// TwinCAT 3 PLC project PLC1
// ProgramVersion: 3.1.4024.0
// libraries:
//   SPT Base Types, * (Beckhoff Automation LLC)
//   SPT Event Logger, * (Beckhoff Automation LLC)
//   Tc2_Standard, * (Beckhoff Automation GmbH)
//   Tc2_System, * (Beckhoff Automation GmbH)
//   Tc3_Module, * (Beckhoff Automation GmbH)
//   XPlanarApplication, * (Beckhoff Automation LLC)
// project tree:
//   / GlobalTextList.TcGTLO, PlcTask.TcTTO, Visualization Manager.TcVMO (not stored)
//   POUs/CustomStations/ FB_RoutingStation.TcPOU, FB_RotateStation.TcPOU
//   POUs/ FB_XPlanarModule.TcPOU, MAIN.TcPOU
//   POUs/Utilities/ ErrorStep.TcPOU (not stored), NextMinorStep.TcPOU (not stored), NextStep.TcPOU
//   VISUs/ V_Main.TcVIS
// real-time tasks:
//   TASK XPlanar Task3: cycle T#250us, priority 1, ADS port 350
//   TASK XPlanar Task4: cycle T#250us, priority 2, ADS port 351
//   TASK XPlanar Task5: cycle T#250us, priority 3, ADS port 352
//   TASK MC-Task (MET): cycle T#2ms, priority 4, ADS port 353
//   TASK MC-Task (MPT): cycle T#10ms, priority 5, ADS port 354
//   TASK Job Task: cycle default, priority 6
//   TASK PlcTask: cycle T#10ms, priority 20, ADS port 355
// variable links:
//   XPlanar MC Project/Axes/Mover4330_1 <-> TcCOM Objects/XPlanar/Mover4330_1
//     McToIo/STD <-> InputsFromNC3/NC3ToHW
//   XPlanar MC Project/Axes/Mover4330_2 <-> TcCOM Objects/XPlanar/Mover4330_2
//     IoToMc/STD <-> OutputsToNC3/HWToNC3
//   XPlanar MC Project/Axes/Mover4330_3 <-> TcCOM Objects/XPlanar/Mover4330_3
//     IoToMc/STD <-> OutputsToNC3/HWToNC3
//   XPlanar MC Project/Axes/Mover4330_4 <-> TcCOM Objects/XPlanar/Mover4330_4
//     IoToMc/STD <-> OutputsToNC3/HWToNC3
//   PLC1/PLC1 Instance <-> XPlanar MC Project/Axes/Mover4330_1
//     PlcTask Inputs/MAIN.XPlanarModule.Mover[1]._Mover.MCTOPLC/ACT <-> McToPlc/ACT
//     PlcTask Inputs/MAIN.XPlanarModule.Mover[1]._Mover.MCTOPLC/COORDMODE <-> McToPlc/COORDMODE
//     PlcTask Inputs/MAIN.XPlanarModule.Mover[1]._Mover.MCTOPLC/SET <-> McToPlc/SET
//     PlcTask Inputs/MAIN.XPlanarModule.Mover[1]._Mover.MCTOPLC/SETONTRACK <-> McToPlc/SETONTRACK
//     PlcTask Inputs/MAIN.XPlanarModule.Mover[1]._Mover.MCTOPLC/STD <-> McToPlc/STD
//     PlcTask Outputs/MAIN.XPlanarModule.Mover[1]._Mover.PLCTOMC/STD <-> PlcToMc/STD
//   PLC1/PLC1 Instance <-> XPlanar MC Project/Axes/Mover4330_2
//     PlcTask Inputs/MAIN.XPlanarModule.Mover[2]._Mover.MCTOPLC/ACT <-> McToPlc/ACT
//     PlcTask Inputs/MAIN.XPlanarModule.Mover[2]._Mover.MCTOPLC/COORDMODE <-> McToPlc/COORDMODE
//     PlcTask Inputs/MAIN.XPlanarModule.Mover[2]._Mover.MCTOPLC/SET <-> McToPlc/SET
//     PlcTask Inputs/MAIN.XPlanarModule.Mover[2]._Mover.MCTOPLC/SETONTRACK <-> McToPlc/SETONTRACK
//     PlcTask Inputs/MAIN.XPlanarModule.Mover[2]._Mover.MCTOPLC/STD <-> McToPlc/STD
//     PlcTask Outputs/MAIN.XPlanarModule.Mover[2]._Mover.PLCTOMC/STD <-> PlcToMc/STD
//   PLC1/PLC1 Instance <-> XPlanar MC Project/Axes/Mover4330_3
//     PlcTask Inputs/MAIN.XPlanarModule.Mover[3]._Mover.MCTOPLC/ACT <-> McToPlc/ACT
//     PlcTask Inputs/MAIN.XPlanarModule.Mover[3]._Mover.MCTOPLC/COORDMODE <-> McToPlc/COORDMODE
//     PlcTask Inputs/MAIN.XPlanarModule.Mover[3]._Mover.MCTOPLC/SET <-> McToPlc/SET
//     PlcTask Inputs/MAIN.XPlanarModule.Mover[3]._Mover.MCTOPLC/SETONTRACK <-> McToPlc/SETONTRACK
//     PlcTask Inputs/MAIN.XPlanarModule.Mover[3]._Mover.MCTOPLC/STD <-> McToPlc/STD
//     PlcTask Outputs/MAIN.XPlanarModule.Mover[3]._Mover.PLCTOMC/STD <-> PlcToMc/STD
//   PLC1/PLC1 Instance <-> XPlanar MC Project/Axes/Mover4330_4
//     PlcTask Inputs/MAIN.XPlanarModule.Mover[4]._Mover.MCTOPLC/ACT <-> McToPlc/ACT
//     PlcTask Inputs/MAIN.XPlanarModule.Mover[4]._Mover.MCTOPLC/COORDMODE <-> McToPlc/COORDMODE
//     PlcTask Inputs/MAIN.XPlanarModule.Mover[4]._Mover.MCTOPLC/SET <-> McToPlc/SET
//     PlcTask Inputs/MAIN.XPlanarModule.Mover[4]._Mover.MCTOPLC/SETONTRACK <-> McToPlc/SETONTRACK
//     PlcTask Inputs/MAIN.XPlanarModule.Mover[4]._Mover.MCTOPLC/STD <-> McToPlc/STD
//     PlcTask Outputs/MAIN.XPlanarModule.Mover[4]._Mover.PLCTOMC/STD <-> PlcToMc/STD
//   PLC1/PLC1 Instance <-> XPlanar MC Project/Groups/Environment
//     PlcTask Inputs/XPlanarApplication.XPlanar.Environment.MCTOPLC_STD <-> McToPlc/STD
//   PLC1/PLC1 Instance <-> XPlanar MC Project/Groups/Track1
//     PlcTask Inputs/MAIN.XPlanarModule.Track[1]._Track.MCTOPLC_STD <-> McToPlc/STD
//   PLC1/PLC1 Instance <-> XPlanar MC Project/Groups/Track2
//     PlcTask Inputs/MAIN.XPlanarModule.Track[2]._Track.MCTOPLC_STD <-> McToPlc/STD
//   PLC1/PLC1 Instance <-> XPlanar MC Project/Groups/Track3
//     PlcTask Inputs/MAIN.XPlanarModule.Track[3]._Track.MCTOPLC_STD <-> McToPlc/STD
//   PLC1/PLC1 Instance <-> XPlanar MC Project/Groups/XPlanar
//     PlcTask Inputs/XPlanarApplication.XPlanar.Group.MCTOPLC_STD <-> McToPlc/STD
//   TcCOM Objects/XPlanar/Mover4330_1 <-> XPlanar MC Project/Axes/Mover4330_1
//     OutputsToNC3/HWToNC3 <-> IoToMc/STD
//   TcCOM Objects/XPlanar/Mover4330_2 <-> XPlanar MC Project/Axes/Mover4330_2
//     InputsFromNC3/NC3ToHW <-> McToIo/STD
//   TcCOM Objects/XPlanar/Mover4330_3 <-> XPlanar MC Project/Axes/Mover4330_3
//     InputsFromNC3/NC3ToHW <-> McToIo/STD
//   TcCOM Objects/XPlanar/Mover4330_4 <-> XPlanar MC Project/Axes/Mover4330_4
//     InputsFromNC3/NC3ToHW <-> McToIo/STD

CONFIGURATION PLC1
    RESOURCE PLC ON TwinCAT3
        TASK PlcTask(INTERVAL := T#10ms, PRIORITY := 20);
        PROGRAM MAIN WITH PlcTask : MAIN;
    END_RESOURCE
END_CONFIGURATION

// ---- POUs/MAIN.TcPOU
PROGRAM MAIN
VAR
	//Main machine module declaration
	XPlanarModule : FB_XPlanarModule;

	//Control Source for running machine
	ControlSourceHMI : FB_ControlSource;
	ControlSourcePB	 : FB_ControlSource;

	//Local Vars
	InitComplete : BOOL;
END_VAR

CyclicLogic();

METHOD CyclicLogic
VAR_INPUT
END_VAR
IF NOT InitComplete THEN
	InitComplete := Initialize();
	RETURN;
END_IF

//Machine support HMI & Production Monitor
ControlSourcePB.CyclicLogic();
ControlSourceHMI.CyclicLogic();

//Machine Cyclic Logic
XPlanarModule.CyclicLogic();
END_METHOD

METHOD Initialize : BOOL
//Top level machine initialization should happen here, in the main initialization METHOD. Each subsequent "layer" OF modules will be named within their respective "parent" intialize METHOD
IF NOT ControlSourceHMI.Registered THEN
	XPlanarModule.RegisterExternalController(ControlSourceHMI);
END_IF

IF NOT ControlSourcePB.Registered THEN
	XPlanarModule.RegisterExternalController(ControlSourcePB);
END_IF

ControlSourceHMI.CyclicLogic();
ControlSourcePB.CyclicLogic();

//ADSLOGSTR(ADSLOG_MSGTYPE_WARN, 'Lag Monitoring disabled', 'For simulation demo only',);
Initialize := TRUE;
END_METHOD

END_PROGRAM

// ---- POUs/FB_XPlanarModule.TcPOU
FUNCTION_BLOCK FB_XPlanarModule EXTENDS FB_PackML_BaseModule
VAR
	// Component definitions here
	XPlanarTable : FB_Component_Xplanar := (Name := 'XPlanarTable');

	//Station Components
	Station1 : FB_RotateStation	 := (Name := 'Station1'); //Declaration of a custom station
	Station2 : FB_RoutingStation := (Name := 'Station2');
	Station3 : FB_RotateStation	 := (Name := 'Station3');
	Station4 : FB_RotateStation	 := (Name := 'Station4');

	//Helper Vars
	Mover			  : ARRAY[1..SystemParameters.MOVER_COUNT] OF FB_XPlanarMover;
	Track			  : ARRAY[1..SystemParameters.TRACK_COUNT] OF FB_XPlanarTrackSegment;
	TracksInitialized : BOOL;
END_VAR

//! @summary This method contains code which will execute when this PackML module is in the <b>Aborting</b> state
METHOD PROTECTED Aborting
VAR
	i				: UDINT;
	SubModulesReady : BOOL := TRUE;
END_VAR
CASE DescendantSequenceState OF
	0:
		NoStateTasksToComplete := FALSE;
		NextStep(DescendantSequenceState);

	10:
		IF XPlanarTable.Abort() THEN
			StateTasksComplete := TRUE;
			NextStep(DescendantSequenceState);
		END_IF

	20:
		StateTasksComplete := TRUE;
END_CASE

SUPER^.Aborting();
END_METHOD

//! @summary This method contains code which will execute when this PackML module is in the <b>Clearing</b> state
METHOD PROTECTED Clearing
VAR
	i				: UDINT;
	SubModulesReady : BOOL := TRUE;
END_VAR

VAR_INST
	ipResult : I_PlanarTaskResult;
END_VAR

(*! <description> <b>Note:</b> The <i>Clear</i> command can also be thought of as a <i>fault reset</i> depite the ambiguity in the naming of the <i>Reset</i> state. 
<table> 
	<tr>
		<th> Previous State </th>
		<th> Transition In </th>
		<th> Transition Out </th>
		<th> Next State  </th> 
	</tr>
	<tr>
		<td> Aborted </td>
		<td> Clear Command </td> 
		<td> State Complete </td>
		<td> Stopped </td> 
	</tr>
</table>
This method is called as required by <c>StateControl()</c>
</description> 

*)
CASE _CurrentMode OF
	E_PMLUnitMode.ePMLUnitMode_Production:
		CASE DescendantSequenceState OF
			0: //Init
				NoStateTasksToComplete := FALSE;

				//Reset Stations
				Station1.Reset();
				Station2.Reset();
				Station3.Reset();
				NextStep(DescendantSequenceState);

			10: //Reset XPlanar System
				IF XPlanarTable.Reset() THEN
					NextStep(DescendantSequenceState);
				END_IF

			20: //Enable Group
				ipResult := XPlanarTable.EnableGroup();
				IF ipResult.Done THEN
					NextStep(DescendantSequenceState);
				ELSIF ipResult.Error THEN
					ErrorStep(DescendantSequenceState);
				END_IF

			30: //Clearing complete			
				StateTasksComplete := TRUE;
		END_CASE

	E_PMLUnitMode.ePMLUnitMode_Manual:
		;
END_CASE

SUPER^.Clearing();
END_METHOD

METHOD CyclicLogic
VAR
	i : INT;
END_VAR
IF NOT _InitComplete THEN
	_InitComplete := Initialize();
END_IF

//Add any required cyclic logic here

//Call the base logic
SUPER^.CyclicLogic();
END_METHOD

//! @summary This method contains code which will execute when this PackML module is in the <b>Execute</b> state
METHOD PROTECTED Execute
VAR
	i : UDINT;
END_VAR
CASE _CurrentMode OF
	E_PMLUnitMode.ePMLUnitMode_Production:
		FOR i := 1 TO SystemParameters.STATION_COUNT DO
			ip.Stations[i].Execute();
		END_FOR

	E_PMLUnitMode.ePMLUnitMode_Manual:
		; //Insert logic for Manual Mode here
END_CASE
END_METHOD

//! @summary Automatically enables and disables HMI control based on the PackML mode
METHOD PROTECTED HMIPermissions

//! @description This method is called cyclically by <c>CyclicLogic()</c>
//General Mode Based Monitoring and handling of HMI control
CASE _CurrentMode OF
	E_PMLUnitMode.ePMLUnitMode_Production:
		AllowHMIControl(ThisModuleOnly := FALSE);

	E_PMLUnitMode.ePMLUnitMode_Manual:
		AllowHMIControl(ThisModuleOnly := FALSE);

	E_PMLUnitMode.ePMLUnitMode_Maintenance:
		AllowHMIControl(ThisModuleOnly := FALSE);
END_CASE
END_METHOD

//! @summary Basic module initialization logic
METHOD PROTECTED Initialize : BOOL;
VAR
	i						 : UDINT;
	varInfo					 : __SYSTEM.VAR_INFO;
	AllSubUnitsInitialized	 : BOOL := TRUE;
	AllComponentsInitialized : BOOL := TRUE;
END_VAR

//! @description This method is called by <c>CyclicLogic()</c> as required
Initialize := FALSE;
CASE DescendantSequenceState OF
	0: //Register Submodules and Components
		RegisterComponent(XPlanarTable);
		RegisterComponent(Station1);
		RegisterComponent(Station2);
		RegisterComponent(Station3);
		RegisterComponent(Station4);
		_LogModeChanges			:= FALSE;
		_LogStateChanges		:= FALSE;
		DescendantSequenceState := DescendantSequenceState + 10;

	10: //Set interfaces *This must be done before initializing the base class!

		//Set mover interfaces
		FOR i := 1 TO SystemParameters.MOVER_COUNT DO
			Mover[i].MoverIndex := i;
			ip.Movers[i]		:= Mover[i];
		END_FOR

		//Set Track Interfaces
		FOR i := 1 TO SystemParameters.TRACK_COUNT DO
			ip.Tracks[i] := Track[i];
		END_FOR

		//Set Station interfaces
		ip.Stations[1]			:= Station1;
		ip.Stations[2]			:= Station2;
		ip.Stations[3]			:= Station3;
		ip.Stations[4]			:= Station4;
		DescendantSequenceState := DescendantSequenceState + 10;

	20: //Call Initialize of the base class
		IF SUPER^.Initialize() THEN
			DescendantSequenceState := DescendantSequenceState + 10;
		END_IF

	30:
		Initialize := TRUE;
END_CASE
END_METHOD

METHOD PROTECTED Resetting
VAR_INST
	i			 : UDINT;
	ipTaskResult : I_PlanarTaskResult;
END_VAR
CASE _CurrentMode OF
	E_PMLUnitMode.ePMLUnitMode_Production:
		CASE DescendantSequenceState OF
			0: //Init
				i					   := 1;
				NoStateTasksToComplete := FALSE;
				NextStep(DescendantSequenceState);

			10: //Enable Tracks
				ipTaskResult := XplanarTable.EnableTracks();
				IF ipTaskResult.Done THEN
					NextStep(DescendantSequenceState);
				ELSIF ipTaskResult.Error THEN //An error occured, jump to 'error step'
					ErrorStep(DescendantSequenceState);
				END_IF

			20: //Enable Movers
				ipTaskResult := XPlanarTable.EnableMovers();
				IF ipTaskResult.Done THEN
					NextStep(DescendantSequenceState);
				ELSIF ipTaskResult.Error THEN //An error occured, jump to 'error step'
					ErrorStep(DescendantSequenceState);
				END_IF

			30: //Add Tracks to Group
				ipTaskResult := XPlanarTable.AddTracksToGroup();
				IF ipTaskResult.Done THEN
					NextStep(DescendantSequenceState);
				ELSIF ipTaskResult.Error THEN //An error occured, jump to 'error step'
					ErrorStep(DescendantSequenceState);
				END_IF

			40: //Add Movers to Group			
				ipTaskResult := XPlanarTable.AddMoversToGroup();
				IF ipTaskResult.Done THEN
					NextStep(DescendantSequenceState);
				ELSIF ipTaskResult.Error THEN //An error occured, jump to 'error step'
					ErrorStep(DescendantSequenceState);
				END_IF

			50: //Clearing complete
				StateTasksComplete := TRUE;
		END_CASE
END_CASE

SUPER^.Resetting();
END_METHOD

METHOD PRIVATE SetupStations : BOOL
VAR_INPUT
END_VAR
//Set Required Process Station Initialization Parameters
Station1.Position.SetValuesXYC(120, 360, 0);
Station1.Size.x		   := 120;		//Changes the station size in the X plane (optional - Default is 120mm)
Station1.Size.y		   := 120;		//Changes the station size in the Y plane (optionsl- Default is 120mm)
Station1.TrackID	   := 1;		//Set Index of the track segment the station resides on if applicable	
Station1.NextStation   := Station2; //Set the interface for the next station of the mover
Station1.StationAngle  := 90;
Station1.NumberOfTurns := 0;

Station2.Position.SetValuesXYC(360, 600, 0);
Station2.StationType := E_StationType.DecisionPoint; //Set type to DecisionPoint for 'on the fly' processing
Station2.OutputA := Station3;
Station2.OutputB := Station4;
Station2.TrackID	   := 1;

Station3.Position.SetValuesXYC(600, 360, 0);
Station3.TrackID	   := 2;
Station3.NextStation   := Station1;
Station3.StationAngle  := 360;
Station3.NumberOfTurns := 1;

Station4.Position.SetValuesXYC(840, 360, 0);
Station4.TrackID	   := 3;
Station4.NextStation   := Station1;
Station4.StationAngle  := -90;
Station4.NumberOfTurns := 0;

//Return TRUE when all necessary station parameters are set
SetupStations := TRUE;
END_METHOD

METHOD PROTECTED Starting
VAR_INST
	i		 : UDINT;
	ipResult : I_PlanarTaskResult;
END_VAR
CASE _CurrentMode OF
	E_PMLUnitMode.ePMLUnitMode_Production:
		CASE DescendantSequenceState OF
			0:
				NoStateTasksToComplete	:= FALSE;
				DescendantSequenceState := 10;
				i						:= 1;

			10: //Set Station Parameters
				SetupStations();
				NextStep(DescendantSequenceState);

			20: //Cleanup mover queues
				FOR i := 1 TO SystemParameters.STATION_COUNT DO
					ip.Stations[i].MoverQueue.Dequeue();
				END_FOR

				NextStep(DescendantSequenceState);

			30: //Set some initial application move dynamics
				FOR i := 1 TO SystemParameters.MOVER_COUNT DO
					ip.Movers[i].Dynamics.Movement.Accel	:= 2000;
					ip.Movers[i].Dynamics.Movement.Decel	:= 2000;
					ip.Movers[i].Dynamics.Movement.Velocity := 300;
					ip.Movers[i].Dynamics.Movement.Jerk		:= 50000;
					ip.Movers[i].Dynamics.Rotation.Accel	:= 5000;
					ip.Movers[i].Dynamics.Rotation.Decel	:= 5000;
					ip.Movers[i].Dynamics.Rotation.Velocity := 300;
					ip.Movers[i].Dynamics.Rotation.Jerk		:= 100000;
					ip.Movers[i].Dynamics.Tilt.Accel		:= 5000;
					ip.Movers[i].Dynamics.Tilt.Decel		:= 5000;
					ip.Movers[i].Dynamics.Tilt.Velocity		:= 300;
					ip.Movers[i].Dynamics.Tilt.Jerk			:= 100000;
					ip.Movers[i].Gap						:= 250;
					ip.Movers[i].Destination				:= 0;
				END_FOR

				i := 1;
				NextStep(DescendantSequenceState);

			40: //Join Movers to nearest track
				IF i <= SystemParameters.MOVER_COUNT THEN
					ipResult := ip.Movers[i].MoveCommand.JoinClosestTrack(FALSE);
					IF ipResult.Done THEN
						NextMinorStep(DescendantSequenceState);
					ELSIF ipResult.Error THEN
						ErrorStep(DescendantSequenceState);
					END_IF
				ELSE
					i := 1;
					NextStep(DescendantSequenceState);
				END_IF

			41: //Check Mover Count
				IF i <= SystemParameters.MOVER_COUNT THEN
					i						:= i + 1;
					DescendantSequenceState := 40;
				ELSE
					i := 1;
					NextStep(DescendantSequenceState);
				END_IF

			50: //Send Movers around to station 1
				IF i <= SystemParameters.MOVER_COUNT THEN
					ipResult := ip.Movers[i].MoveCommand.SendToStation(ip.Stations[1]);
					IF ipResult.Busy THEN
						NextMinorStep(DescendantSequenceState);
					ELSIF ipResult.Error THEN
						ErrorStep(DescendantSequenceState);
					END_IF
				ELSE
					i := 1;
					NextStep(DescendantSequenceState);
				END_IF

			51: //Check Mover Count
				IF i <= SystemParameters.MOVER_COUNT THEN
					i						:= i + 1;
					DescendantSequenceState := 50;
				ELSE
					i := 1;
					NextStep(DescendantSequenceState);
				END_IF

			60:
				StateTasksComplete := TRUE;
		END_CASE

	E_PMLUnitMode.ePMLUnitMode_Manual:
		;
END_CASE

SUPER^.Starting();
END_METHOD

END_FUNCTION_BLOCK

// ---- POUs/CustomStations/FB_RotateStation.TcPOU
FUNCTION_BLOCK FB_RotateStation EXTENDS FB_XPlanarStationBase
VAR
	_StationAngle  : LREAL;
	_NumberOfTurns : DINT;
END_VAR

METHOD Execute
VAR_INST
	i			  : UDINT := 1;
	CommandResult : I_PlanarTaskResult;
END_VAR
SUPER^.Execute();
IF StationState = E_XPlanarStationState.ProcessMover THEN
	CommandResult := ipCurrentMover.MoveCommand.Rotate(_StationAngle, _NumberOfTurns);
	IF CommandResult.Done THEN
		_StationComplete := TRUE;
	ELSIF CommandResult.Error THEN
		; //Command returned an error!
	END_IF
END_IF
END_METHOD

PROPERTY NumberOfTurns : DINT
SET
_NumberOfTurns := NumberOfTurns;
END_SET
END_PROPERTY

PROPERTY StationAngle : LREAL
SET
_StationAngle := StationAngle;
END_SET
END_PROPERTY

END_FUNCTION_BLOCK

// ---- POUs/CustomStations/FB_RoutingStation.TcPOU
FUNCTION_BLOCK FB_RoutingStation EXTENDS FB_XPlanarStationBase
VAR_INPUT
END_VAR
VAR_OUTPUT
END_VAR
VAR
	_OutputA	: I_XplanarStation;
	_OutputB	: I_XPlanarStation;
END_VAR

METHOD Execute
SUPER^.Execute(); //Call the base station logic to handle sending and receiving of movers

//When the station is in the Process mover state you can perform any application specific station logic
IF StationState = E_XPlanarStationState.ProcessMover THEN
	IF _OutputA <> 0 AND _OutputB <> 0 THEN	
		CASE ipCurrentMover.MoverIndex OF
			1, 3:
				ipNextStation := _OutputA;
			2, 4:
				ipNextStation := _OutputB;
		END_CASE
		
		_StationComplete := TRUE;	//Set _StationComplete TRUE when done.  This will be automatically reset when the mover exits
	END_IF
END_IF
END_METHOD

PROPERTY OutputA : I_XPlanarStation
SET
_OutputA := OutputA;
END_SET
END_PROPERTY

PROPERTY OutputB : I_XPlanarStation
SET
_OutputB := OutputB;
END_SET
END_PROPERTY

END_FUNCTION_BLOCK

// ---- POUs/Utilities/NextStep.TcPOU
FUNCTION NextStep : UDINT
VAR_IN_OUT
	StateVar : UDINT;
END_VAR

NextStep := StateVar := ((StateVar / 10) * 10) + 10;

END_FUNCTION

// ---- GlobalTextList.TcGTLO
TEXTLIST GlobalTextList
  944 = 'HMI PB Station'
  924 = 'Pushbutton Station'
  181 = 'Reset'
  77 = 'Start'
  828 = 'Stop'
END_TEXTLIST

// ---- VISUs/V_Main.TcVIS
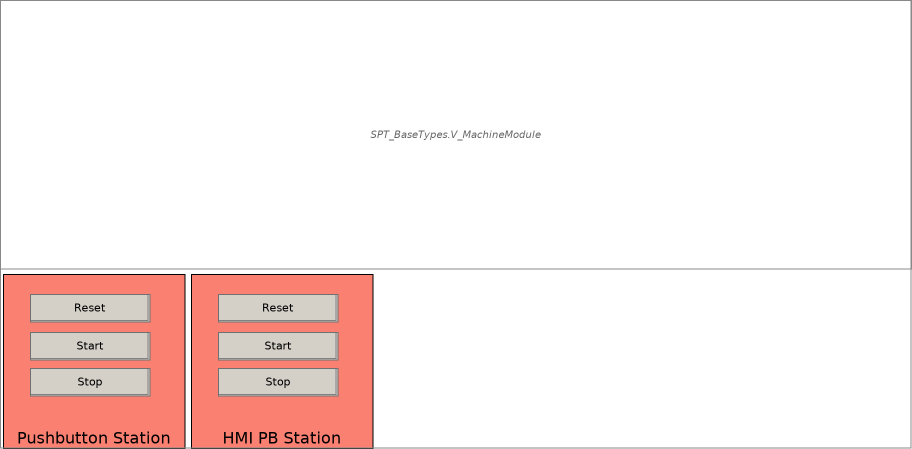
VISUALIZATION V_Main  // 912x449
    Frame (0,0 912x269)
        shows SPT_BaseTypes.V_MachineModule(HMI := MAIN.XPlanarModule.PackMLBaseModule_HMI)
    Group (3,274 182x175)
        RoundedRectangle (0,0 182x175), "Pushbutton Station"
        Button (27,94 120x28), "Stop", input disabled if: not MAIN.ControlSourcePB.MainPMLControl_Simplified.StopPermissive
            tap MAIN.ControlSourcePB.MainPMLControl_Simplified.StopPressed
        Button (27,20 120x28), "Reset", input disabled if: not MAIN.ControlSourcePB.MainPMLControl_Simplified.ResetPermissive
            tap MAIN.ControlSourcePB.MainPMLControl_Simplified.ResetPressed
        Button (27,58 120x28), "Start", input disabled if: not MAIN.ControlSourcePB.MainPMLControl_Simplified.StartPermissive
            tap MAIN.ControlSourcePB.MainPMLControl_Simplified.StartPressed
    Group (191,274 182x175)
        RoundedRectangle (0,0 182x175), "HMI PB Station"
        Button (27,94 120x28), "Stop", input disabled if: not MAIN.ControlSourceHMI.MainPMLControl_Simplified.StopPermissive
            tap MAIN.ControlSourceHMI.MainPMLControl_Simplified.StopPressed
        Button (27,20 120x28), "Reset", input disabled if: not MAIN.ControlSourceHMI.MainPMLControl_Simplified.ResetPermissive
            tap MAIN.ControlSourceHMI.MainPMLControl_Simplified.ResetPressed
        Button (27,58 120x28), "Start", input disabled if: not MAIN.ControlSourceHMI.MainPMLControl_Simplified.StartPermissive
            tap MAIN.ControlSourceHMI.MainPMLControl_Simplified.StartPressed
END_VISUALIZATION
